TYPE sysOutputs :
STRUCT
	
	oAlarm		AT %Q*: BOOL;
	oCloseDoor	AT %Q*: BOOL;
	oOpenDoor	AT %Q*: BOOL;
	
	// MOTOR NEMA17 / TB6600
    oMotorPulse AT %Q*: BOOL;   // → PUL- del TB6600
    oMotorDir   AT %Q*: BOOL;   // → DIR- del TB6600

	//
	oLightGreen  : BOOL;
	oLightOrange : BOOL;
	oLightRed    : BOOL;

	
END_STRUCT
END_TYPE

(* stored: Version 1.1.0.1, ProductVersion 3.1.4026.12
   DUT sysOutputs: Id {50a3c6c6-ca5f-40b2-876c-d6ede982efb7} *)
